FUNCTION_BLOCK ObjectRunner EXTENDS CyclicBase IMPLEMENTS I_ObjectRunner
VAR_INPUT
END_VAR
VAR_OUTPUT
END_VAR
VAR
	CyclicModules : ARRAY[0..MaxRegisteredModules] OF ICyclic;
	ModuleCount : INT := 0;
	InitModuleCount : INT := 0;
	InitialiseModules : ARRAY[0..MaxRegisteredModules] OF I_Initialise;
	i: INT;
	InitialisationCount : INT := 0;
	Registered: BOOL;
	Initialised : BOOL := FALSE;
END_VAR
VAR CONSTANT
	MaxRegisteredModules : INT := 99;
END_VAR

METHOD AreAllModuleInitialised : BOOL
VAR_INPUT
END_VAR
AreAllModuleInitialised := Initialised;
END_METHOD

METHOD PUBLIC  Cycle : HRESULT
VAR_INPUT
END_VAR
IF Initialised THEN
	FOR i := 0 TO MaxRegisteredModules DO
		IF CyclicModules[i] <> 0 THEN
			CyclicModules[i].Cycle();
		END_IF
	END_FOR
END_IF
END_METHOD

METHOD DeregisterAllModules : HRESULT
VAR_INPUT
END_VAR
FOR i := 0 TO MaxRegisteredModules DO
	CyclicModules[i] := 0;
	InitialiseModules[i] := 0;
END_FOR
ModuleCount := 0;
InitModuleCount := 0;
DeregisterAllModules := S_OK;
END_METHOD

METHOD DeregisterModule : HRESULT
vAR_INPUT
	CyclicModule : ICyclic;
END_VAR
IF ModuleCount > 0 THEN
	DeregisterModule := E_FAIL;
	FOR i := 0 TO ModuleCount DO 
		IF CyclicModules[i] = CyclicModule THEN
			CyclicModules[i] := 0;
			IF InitialiseModules[i] <> 0 THEN
				InitialiseModules[i] := 0;
				InitModuleCount := InitModuleCount - 1;
			END_IF
			ModuleCount := ModuleCount - 1;
			DeregisterModule := 2;
		END_IF
	END_FOR
ELSE
	DeregisterModule := -1;
END_IF
END_METHOD

METHOD GetCyclicModuleCount : INT
VAR_INPUT
END_VAR
GetCyclicModuleCount := ModuleCount;
END_METHOD

METHOD GetInitModuleCount : INT
VAR_INPUT
END_VAR
GetInitModuleCount := InitModuleCount;
END_METHOD

METHOD Initialise : HRESULT
VAR_INPUT
END_VAR
IF InitialisationCount = 0 THEN
	Initialised := TRUE;
	Initialise := S_FALSE;
ELSE
	IF InitialisationCount < MaxRegisteredModules THEN
		IF InitialiseModules[InitialisationCount] <> 0 THEN
			IF InitialiseModules[InitialisationCount].Initialise() = 2 THEN
				InitialisationCount := InitialisationCount + 1;
			END_IF
		ELSE
			InitialisationCount := InitialisationCount + 1;
		END_IF
	ELSE
		Initialise := S_OK;
		InitialisationCount := 0;
		Initialised := TRUE;
	END_IF
END_IF
END_METHOD

METHOD RegisterModule : HRESULT
VAR_INPUT
	CyclicModule : ICyclic;
END_VAR
VAR
	InitInterface : I_Initialise;
END_VAR
IF CyclicModule <> 0 AND_THEN ModuleCount < (MaxRegisteredModules + 1) THEN
	Registered := FALSE;
	FOR i := 0 TO MaxRegisteredModules DO
		IF CyclicModules[i] = CyclicModule THEN
			Registered := TRUE;
		END_IF
	END_FOR
	IF NOT Registered THEN	
		FOR i := 0 TO MaxRegisteredModules DO
			IF CyclicModules[i] = 0 THEN
				CyclicModules[i] := CyclicModule;
				IF __QUERYINTERFACE(CyclicModule,InitInterface) THEN
					InitialiseModules[i] := InitInterface;
					InitModuleCount := InitModuleCount + 1;
				END_IF
				EXIT;
			END_IF
		END_FOR
		ModuleCount := ModuleCount + 1;
		RegisterModule := S_OK;
	ELSE
		RegisterModule := -1;
	END_IF	
ELSE
	RegisterModule := -2;
END_IF
END_METHOD

END_FUNCTION_BLOCK

(* stored: Version 1.1.0.1
   POU ObjectRunner: Id {4adb75ec-914c-46a2-96a4-b49d6ed1e005}, SpecialFunc None
   Method AreAllModuleInitialised: Id {4d383a02-46c6-4353-8362-547fa2f80ae1}
   Method Cycle: Id {07b170dc-1426-48b0-b328-82870c7027f5}
   Method DeregisterAllModules: Id {801399c7-4ed5-4baa-bb84-25ca1ab9b024}
   Method DeregisterModule: Id {dfa8fa7b-42f3-4591-8ff7-fdf50b44b36a}
   Method GetCyclicModuleCount: Id {ce16b2d3-0e8a-4df6-aa9c-1c1b403838ba}
   Method GetInitModuleCount: Id {a9fb930d-907c-4894-834e-3a7f560764dd}
   Method Initialise: Id {498dbf2f-31fd-468f-af2a-ef254d08806c}
   Method RegisterModule: Id {5f816535-6603-4c30-b42c-afe250745821} *)
